FUNCTION ATAN2 : LREAL
VAR_INPUT
	y : LREAL;
	x : LREAL;
END_VAR
VAR
END_VAR

IF (x > 0.0) THEN
	// (x > 0)
	ATAN2 := 2*ATAN(y/(SQRT(EXPT(x, 2.0) + EXPT(y, 2.0)) + x));
ELSIF (y <> 0.0) THEN
	// (x <= 0) & (y != 0)
	ATAN2 := 2*ATAN((SQRT(EXPT(x, 2.0) + EXPT(y, 2.0)) - x)/y);
ELSIF (x < 0.0) THEN
	// (x < 0) & (y == 0)
	ATAN2 := PI;
ELSE
	// (x == 0) & (y == 0) Technically undefined, but we set it to zero
	ATAN2 := 0.0;
END_IF

END_FUNCTION

(* stored: Version 1.1.0.1, ProductVersion 3.1.4024.9
   POU ATAN2: Id {f98b14fc-3cbb-4106-9d71-c37dc554b494}, SpecialFunc None *)
